FUNCTION FUN_ConvFourByteToInt32 : DINT
VAR_INPUT
	nValue1		:BYTE;				// Input Byte no 1
	nValue2		:BYTE;				// Input Byte no 2
	nValue3		:BYTE;				// Input Byte no 3
	nValue4		:BYTE;				// Input Byte no 4
END_VAR
VAR
	uData		:U_Convert_INT32;		// Data variable used for conversion
END_VAR


// Save input bytes in data union
uData.arrByte[1] := nValue1;
uData.arrByte[2] := nValue2;
uData.arrByte[3] := nValue3;
uData.arrByte[4] := nValue4;

// Return value
FUN_ConvFourByteToInt32 := uData.nValue;

END_FUNCTION

(* stored: Version 1.1.0.1, ProductVersion 3.1.4024.12
   POU FUN_ConvFourByteToInt32: Id {ac6a0a79-b0c0-41d6-8b01-cdc0a83d84b9}, SpecialFunc None *)
